// TIA Portal project "Kağıt Ambalaj Konik PLC (1,2,3,4,5)_V15.1" (V15.1)

(* hardware
DEVICE "S7-1200 station_1"  S7-1200 Station
   slot 0: "Rack_0"  S7-1200 Rack  Rack  V1.0
   slot 1: "PLC_1"  CPU 1215C DC/DC/DC  6ES7 215-1AG40-0XB0  V4.2
   slot 2: "DI 16x24VDC_1"  6ES7 221-1BH32-0XB0  V2.0
   slot 3: "AI 8x13BIT_1"  6ES7 231-4HF32-0XB0  V2.0
*)

// ===== PLC "PLC_1"  CPU 1215C DC/DC/DC =====

VAR_GLOBAL   // PLC tag table "Default tag table"
   "Konik 5 Count Value" AT %ID1000 : DWord;
   "Konik 4 Count Value" AT %ID1004 : DWord;
   "Konik 3 Count Value" AT %ID1008 : DWord;
   "Konik 2 Count Value" AT %ID1012 : DWord;
   "Konik 1 Count Value" AT %ID1016 : DWord;
   "Konik 1 Adet Sayaç" AT %I8.4 : Bool;
   "Konik 2 Adet Sayaç" AT %I8.5 : Bool;
   "System_Byte" AT %MB1 : Byte;
   "FirstScan" AT %M1.0 : Bool;
   "DiagStatusUpdate" AT %M1.1 : Bool;
   "AlwaysTRUE" AT %M1.2 : Bool;
   "AlwaysFALSE" AT %M1.3 : Bool;
   "Clock_Byte" AT %MB0 : Byte;
   "Clock_10Hz" AT %M0.0 : Bool;
   "Clock_5Hz" AT %M0.1 : Bool;
   "Clock_2.5Hz" AT %M0.2 : Bool;
   "Clock_2Hz" AT %M0.3 : Bool;
   "Clock_1.25Hz" AT %M0.4 : Bool;
   "Clock_1Hz" AT %M0.5 : Bool;
   "Clock_0.625Hz" AT %M0.6 : Bool;
   "Clock_0.5Hz" AT %M0.7 : Bool;
   "Konik 4 Adet Sayaç" AT %I9.1 : Bool;
   "Konik 5 Adet Sayaç" AT %I9.2 : Bool;
   "Konik 1 Run Bilgisi" AT %I9.3 : Bool;
   "Konik 2 Run Bilgisi" AT %I9.4 : Bool;
   "Konik 3 Run Bilgisi" AT %I9.5 : Bool;
   "Konik 4 Run Bilgisi" AT %I9.6 : Bool;
   "Konik 5 Run Bilgisi" AT %I9.7 : Bool;
   "Konik 3 Adet Sayaç" AT %I9.0 : Bool;
   "Tag_1" AT %M20.0 : Bool;
   "Tag_2" AT %M20.1 : Bool;
   "Tag_3" AT %M20.3 : Bool;
   "Tag_4" AT %M20.4 : Bool;
   "Tag_5" AT %M20.5 : Bool;
   "Tag_6" AT %M20.6 : Bool;
   "Tag_7" AT %M20.7 : Bool;
   "Tag_8" AT %M21.0 : Bool;
   "Tag_test" AT %I0.5 : Bool;
END_VAR

VAR_GLOBAL   // PLC tag table "Tag table_1"
   "Tag_rst_1" AT %M21.1 : Bool;
   "Tag_rst_2" AT %M21.2 : Bool;
   "Tag_rst_3" AT %M21.3 : Bool;
   "Tag_rst_4" AT %M21.5 : Bool;
   "Tag_rst_5" AT %M21.6 : Bool;
   "Tag_rst_6" AT %M21.7 : Bool;
   "Tag_rst_7" AT %M22.0 : Bool;
   "Tag_rst_8" AT %M22.1 : Bool;
   "Tag_rst_9" AT %M22.4 : Bool;
   "Tag_rst_10" AT %M22.5 : Bool;
   "Tag_rst_11" AT %M22.6 : Bool;
   "Tag_rst_12" AT %M22.7 : Bool;
   "Tag_rst_13" AT %M22.3 : Bool;
   "Tag_rst_14" AT %M22.2 : Bool;
   "Tag_rst_15" AT %M21.4 : Bool;
   "Tag_rst_16" AT %M23.0 : Bool;
   "Tag_rst_17" AT %M23.1 : Bool;
   "Tag_rst_18" AT %M23.2 : Bool;
   "Tag_rst_19" AT %M23.3 : Bool;
   "Tag_rst_20" AT %M23.4 : Bool;
   "Tag_rst_21" AT %M23.5 : Bool;
   "Tag_rst_22" AT %M23.6 : Bool;
   "Tag_rst_23" AT %M23.7 : Bool;
   "Tag_rst_24" AT %M24.0 : Bool;
   "hızcontrol" AT %M24.1 : Bool;
   "hızcontrol(1)" AT %M24.2 : Bool;
   "hızcontrol(2)" AT %M24.3 : Bool;
   "hızcontrol(3)" AT %M24.4 : Bool;
   "hızcontrol(4)" AT %M24.5 : Bool;
END_VAR

DATA_BLOCK "DataMeter"   // DB3
{ S7_Optimized_Access := 'FALSE' }
VERSION : 0.1
   VAR
      "Konik 1 Metre Sayac" : UDInt;
      "Konik 2 Metre Sayac" : UDInt;
      "Konik 3 Metre Sayac" : UDInt;
      "Konik 4 Metre Sayac" : UDInt;
      "Konik 5 Metre Sayac" : UDInt;
      "Konik 1 Metre RST" : Bool;
      "Konik 2 Metre RST" : Bool;
      "Konik 3 Metre RST" : Bool;
      "Konik 4 Metre RST" : Bool;
      "Konik 5 Metre RST" : Bool;
      "Konik 1 Hız" : Real;
      "Konik 2 Hız" : Real;
      "Konik 3 Hız" : Real;
      "Konik 4 Hız" : Real;
      "Konik 5 Hız" : Real;
      MultiplierValue : Real := 0.39284;
      EncoderRawValues : Array[0..4] of UDInt;
      TempMeters : Array[0..9] of UDInt;
      Rawspeed : Array[0..7] of Real;
      RealMeterValue : Array[0..7] of Real;
   END_VAR
BEGIN
END_DATA_BLOCK

DATA_BLOCK "DataSteam"   // DB4
{ S7_Optimized_Access := 'FALSE' }
VERSION : 0.1
   VAR
      sayıcıtest : UDInt := 0;
      wordtest : Word;
      udinttest : UDInt;
      dinttest : DInt;
      inttest_1 : Int;
      floattest : Real;
   END_VAR
BEGIN
END_DATA_BLOCK

DATA_BLOCK "DataDI"   // DB5
{ S7_Optimized_Access := 'FALSE' }
VERSION : 0.1
   VAR
      "Konik 1 Üretim sayacı" : UDInt;
      "Konik 2 Üretim sayacı" : UDInt;
      "Konik 3 Üretim sayacı" : UDInt;
      "Konik 4 Üretim sayacı" : UDInt;
      "Konik 5 Üretim sayacı" : UDInt;
      "Konik 1 Besleme Run Sinyal" : Bool;
      "Konik 2 Besleme Run Sinyal" : Bool;
      "Konik 3  BeslemeRun Sinyal" : Bool;
      "Konik 4  BeslemeRun Sinyal" : Bool;
      "Konik 5  BeslemeRun Sinyal" : Bool;
      "Konik 1 Sayac RST" : Bool;
      "Konik 2 Sayac RST" : Bool;
      "Konik 3 Sayac RST" : Bool;
      "Konik 4 Sayac RST" : Bool;
      "Konik 5 Sayac RST" : Bool;
      "Konik 1 Üretim Sayac Hızı" : Int;
      "Konik 2 Üretim Sayac Hızı" : Int;
      "Konik 3 Üretim Sayac Hızı" : Int;
      "Konik 4 Üretim Sayac Hızı" : Int;
      "Konik 5 Üretim Sayac Hızı" : Int;
      "Konik 1 Run Sinyal" : Bool;
      "Konik 2 Run Sinyal" : Bool;
      "Konik 3 Run Sinyal" : Bool;
      "Konik 4 Run Sinyal" : Bool;
      "Konik 5 Run Sinyal" : Bool;
      "Konik RST" : Array[0..9] of Bool;
      "Konik adet temp" : Array[0..9] of UDInt;
      Dakikareset : Bool;
   END_VAR
BEGIN
END_DATA_BLOCK

DATA_BLOCK "DataSendDI"   // DB6
{ S7_Optimized_Access := 'FALSE' }
VERSION : 0.1
   VAR
      "Konik 1 Run Sinyal" : Bool;
      "Konik 2 Run Sinyal" : Bool;
      "Konik 3 Run Sinyal" : Bool;
      "Konik 4 Run Sinyal" : Bool;
      "Konik 5 Run Sinyal" : Bool;
      "Konik 1 Sayac RST" : Bool;
      "Konik 2 Sayac RST" : Bool;
      "Konik 3 Sayac RST" : Bool;
      "Konik 4 Sayac RST" : Bool;
      "Konik 5 Sayac RST" : Bool;
      "Konik 1 Besleme Run Sinyal" : Bool;
      "Konik 2 Besleme Run Sinyal" : Bool;
      "Konik 3  BeslemeRun Sinyal" : Bool;
      "Konik 4  BeslemeRun Sinyal" : Bool;
      "Konik 5  BeslemeRun Sinyal" : Bool;
      "Konik 1 Metre RST" : Bool;
      "Konik 3 Metre RST" : Bool;
      "Konik 4 Metre RST" : Bool;
      "Konik 5 Metre RST" : Bool;
      "Konik 2 Metre RST" : Bool;
      "Konik 1 Üretim sayacı" : Real;
      "Konik 2 Üretim sayacı" : Real;
      "Konik 3 Üretim sayacı" : Real;
      "Konik 4 Üretim sayacı" : Real;
      "Konik 5 Üretim sayacı" : Real;
      "Konik 1 Üretim Sayac Hızı" : Real;
      "Konik 2 Üretim Sayac Hızı" : Real;
      "Konik 3 Üretim Sayac Hızı" : Real;
      "Konik 4 Üretim Sayac Hızı" : Real;
      "Konik 5 Üretim Sayac Hızı" : Real;
      "Konik 1 Metre Sayac" : Real;
      "Konik 2 Metre Sayac" : Real;
      "Konik 3 Metre Sayac" : Real;
      "Konik 4 Metre Sayac" : Real;
      "Konik 5 Metre Sayac" : Real;
      "Konik 1 Hız" : Real;
      "Konik 2 Hız" : Real;
      "Konik 3 Hız" : Real;
      "Konik 4 Hız" : Real;
      "Konik 5 Hız" : Real;
      PLCLiveBit : Real;
   END_VAR
BEGIN
END_DATA_BLOCK

// folder: System blocks/Program resources

DATA_BLOCK "Counter_dakika"   // DB1
{ S7_Optimized_Access := 'TRUE' }
AUTHOR : Simatic
FAMILY : IEC
NAME : CNTR
VERSION : 1.0
// stored: InstanceOfName IEC_COUNTER
"IEC_COUNTER"
BEGIN
END_DATA_BLOCK

DATA_BLOCK "IEC_Counter_0_DB_5"   // DB2
{ S7_Optimized_Access := 'TRUE' }
AUTHOR : Simatic
FAMILY : IEC
NAME : UDCNTR
VERSION : 1.2
// stored: InstanceOfName IEC_UDCOUNTER
"IEC_UDCOUNTER"
BEGIN
END_DATA_BLOCK

DATA_BLOCK "livetimer"   // DB7
{ S7_Optimized_Access := 'TRUE' }
AUTHOR : Simatic
FAMILY : IEC
NAME : IEC_TMR
VERSION : 1.0
// stored: InstanceOfName IEC_TIMER
"IEC_TIMER"
BEGIN
END_DATA_BLOCK

DATA_BLOCK "IEC_Counter_0_DB"   // DB30
{ S7_Optimized_Access := 'TRUE' }
AUTHOR : Simatic
FAMILY : IEC
NAME : UDCNTR
VERSION : 1.2
// stored: InstanceOfName IEC_UDCOUNTER
"IEC_UDCOUNTER"
BEGIN
END_DATA_BLOCK

DATA_BLOCK "IEC_Counter_0_DB_1"   // DB31
{ S7_Optimized_Access := 'TRUE' }
AUTHOR : Simatic
FAMILY : IEC
NAME : UDCNTR
VERSION : 1.2
// stored: InstanceOfName IEC_UDCOUNTER
"IEC_UDCOUNTER"
BEGIN
END_DATA_BLOCK

DATA_BLOCK "IEC_Counter_0_DB_2"   // DB32
{ S7_Optimized_Access := 'TRUE' }
AUTHOR : Simatic
FAMILY : IEC
NAME : UDCNTR
VERSION : 1.2
// stored: InstanceOfName IEC_UDCOUNTER
"IEC_UDCOUNTER"
BEGIN
END_DATA_BLOCK

DATA_BLOCK "IEC_Counter_0_DB_3"   // DB33
{ S7_Optimized_Access := 'TRUE' }
AUTHOR : Simatic
FAMILY : IEC
NAME : UDCNTR
VERSION : 1.2
// stored: InstanceOfName IEC_UDCOUNTER
"IEC_UDCOUNTER"
BEGIN
END_DATA_BLOCK

DATA_BLOCK "IEC_Counter_0_DB_4"   // DB34
{ S7_Optimized_Access := 'TRUE' }
AUTHOR : Simatic
FAMILY : IEC
NAME : UDCNTR
VERSION : 1.2
// stored: InstanceOfName IEC_UDCOUNTER
"IEC_UDCOUNTER"
BEGIN
END_DATA_BLOCK

// folder: (top level)

FUNCTION "EncoderSingleton" : Void   // FC1, LAD
{ S7_Optimized_Access := 'TRUE' }
VERSION : 0.1
   VAR_TEMP   // added for the SCL form of the ladder/FBD networks
      _w1 : Bool;
      _w2 : Bool;
      _w3 : Bool;
      _w4 : Bool;
      _w5 : Bool;
   END_VAR
BEGIN

REGION Network 1: HSC INIT
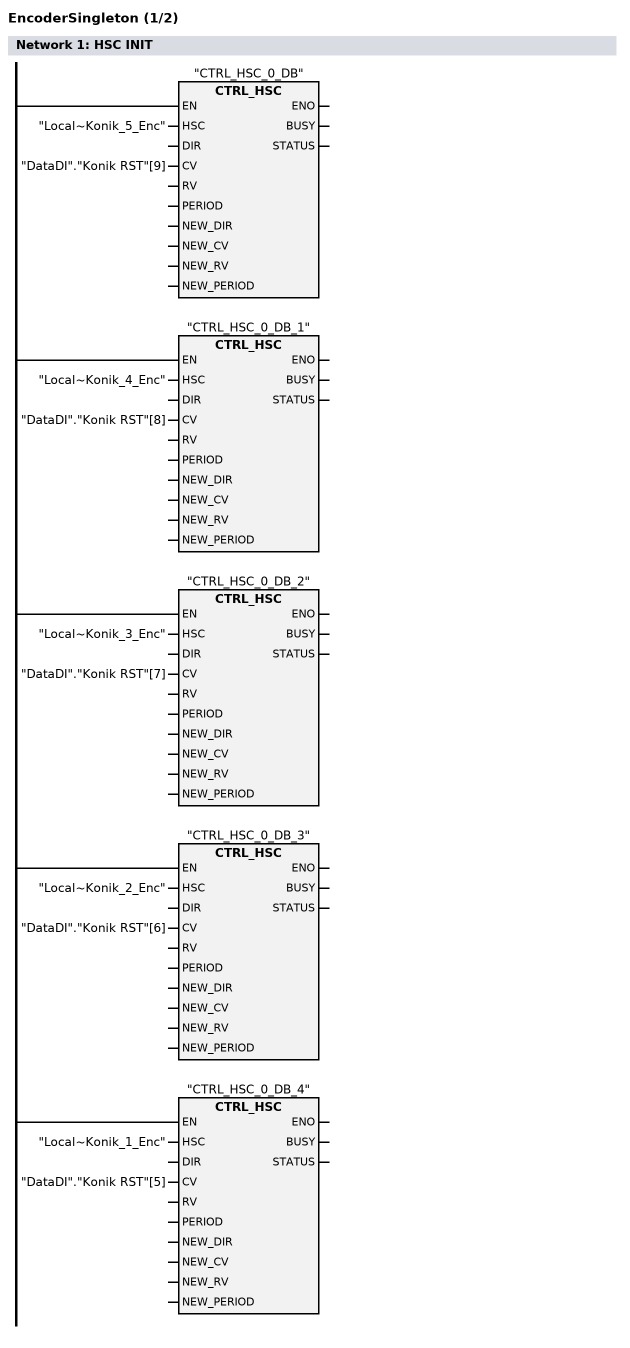
   "CTRL_HSC_0_DB"(HSC := "Local~Konik_5_Enc", CV := "DataDI"."Konik RST"[9]);   // CTRL_HSC
   "CTRL_HSC_0_DB_1"(HSC := "Local~Konik_4_Enc", CV := "DataDI"."Konik RST"[8]);   // CTRL_HSC
   "CTRL_HSC_0_DB_2"(HSC := "Local~Konik_3_Enc", CV := "DataDI"."Konik RST"[7]);   // CTRL_HSC
   "CTRL_HSC_0_DB_3"(HSC := "Local~Konik_2_Enc", CV := "DataDI"."Konik RST"[6]);   // CTRL_HSC
   "CTRL_HSC_0_DB_4"(HSC := "Local~Konik_1_Enc", CV := "DataDI"."Konik RST"[5]);   // CTRL_HSC
END_REGION

REGION Network 2
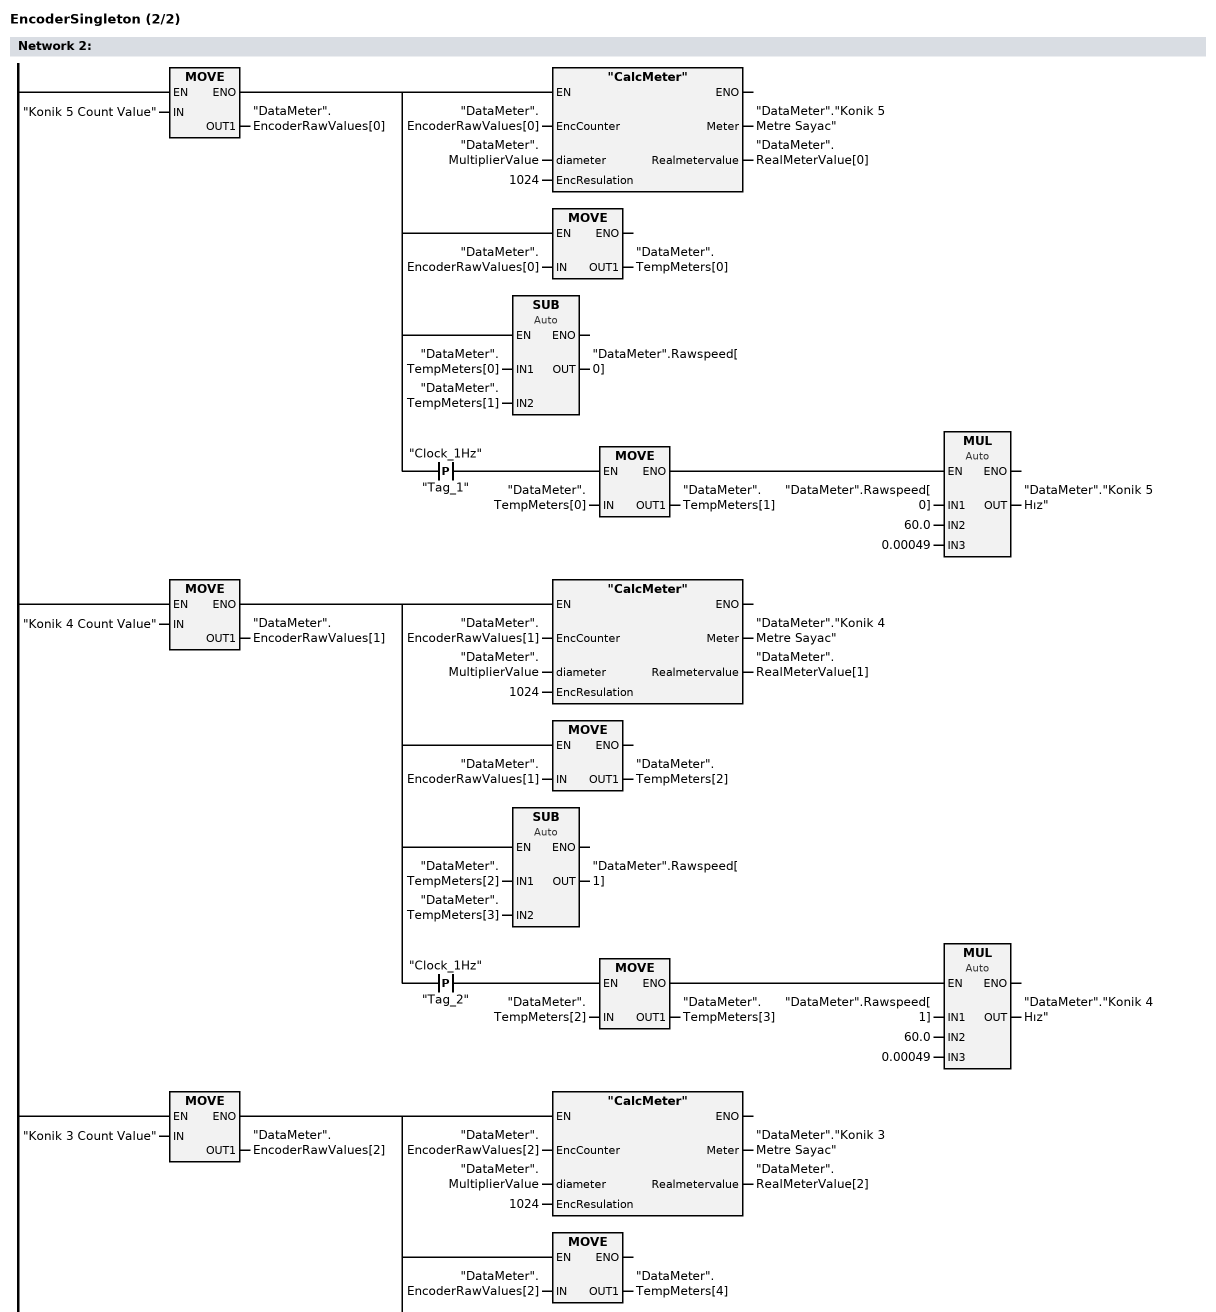
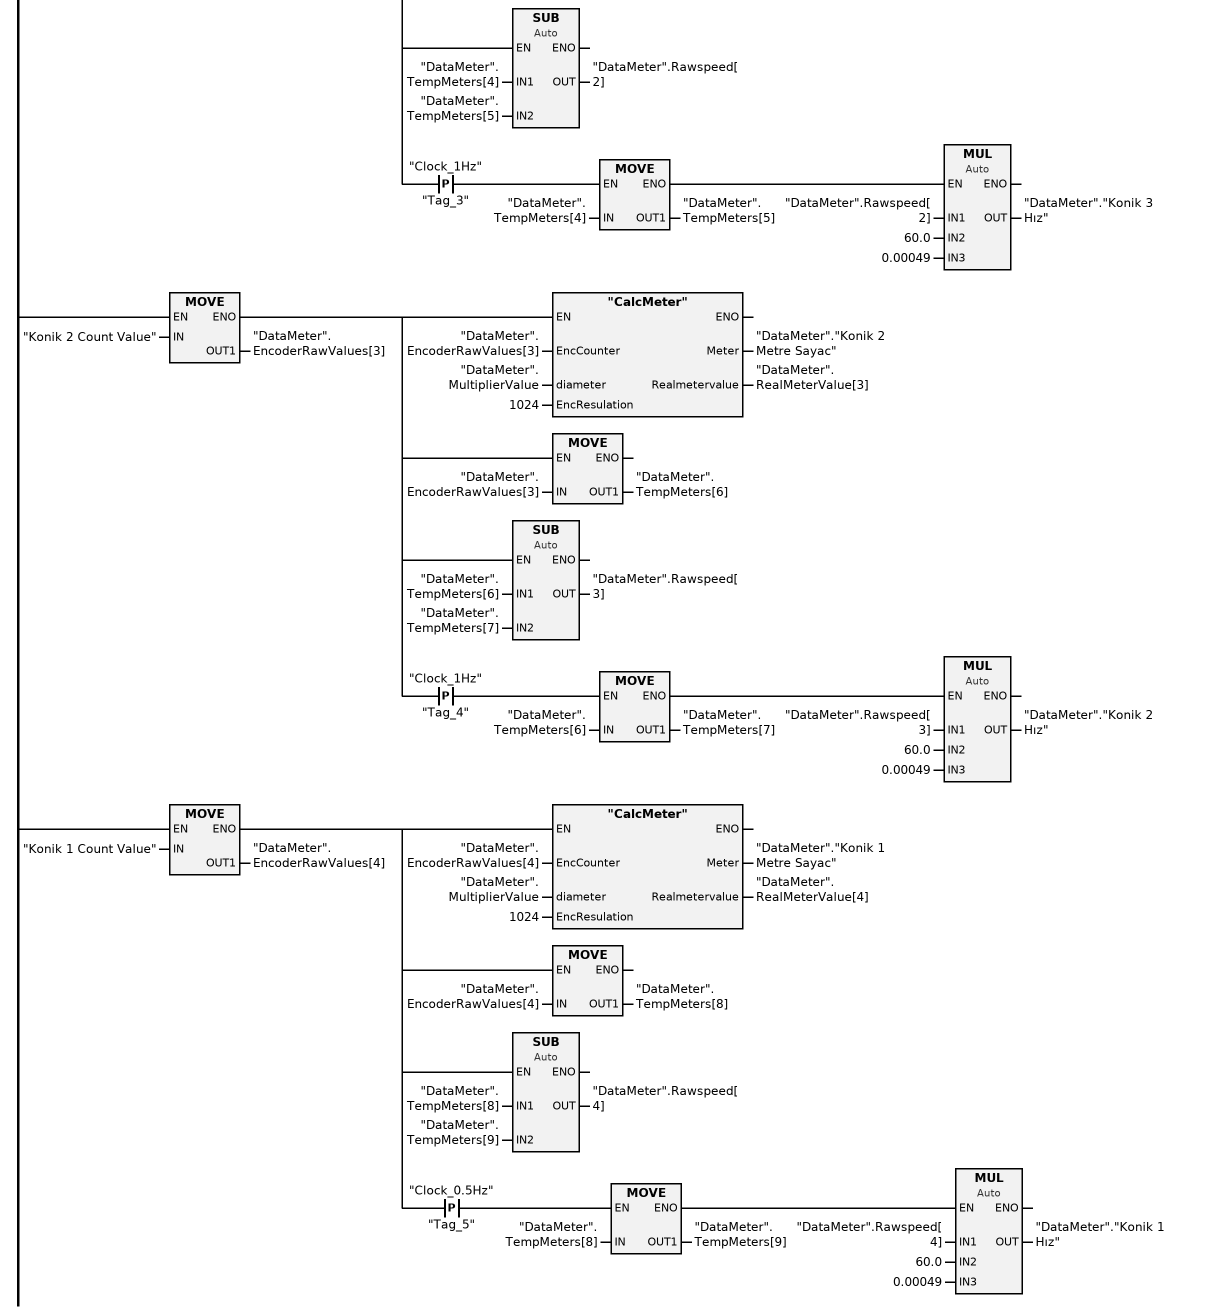
   RUNG wire#powerrail
      Move(in := "Konik 5 Count Value", out1 => "DataMeter".EncoderRawValues[0])
      wire#w1
      "CalcMeter"(EncCounter := "DataMeter".EncoderRawValues[0], diameter := "DataMeter".MultiplierValue, EncResulation := 1024, Meter => "DataMeter"."Konik 5 Metre Sayac", Realmetervalue => "DataMeter".RealMeterValue[0])
   END_RUNG
   RUNG wire#w1
      Move(in := "DataMeter".EncoderRawValues[0], out1 => "DataMeter".TempMeters[0])
   END_RUNG
   RUNG wire#w1
      Sub(in1 := "DataMeter".TempMeters[0], in2 := "DataMeter".TempMeters[1], out => "DataMeter".Rawspeed[0])
   END_RUNG
   RUNG wire#w1
      P_Contact(operand := "Clock_1Hz", bit := "Tag_1")
      Move(in := "DataMeter".TempMeters[0], out1 => "DataMeter".TempMeters[1])
      Mul(in1 := "DataMeter".Rawspeed[0], in2 := 60.0, in3 := 0.00049, out => "DataMeter"."Konik 5 Hız")
   END_RUNG
   RUNG wire#powerrail
      Move(in := "Konik 4 Count Value", out1 => "DataMeter".EncoderRawValues[1])
      wire#w2
      "CalcMeter"(EncCounter := "DataMeter".EncoderRawValues[1], diameter := "DataMeter".MultiplierValue, EncResulation := 1024, Meter => "DataMeter"."Konik 4 Metre Sayac", Realmetervalue => "DataMeter".RealMeterValue[1])
   END_RUNG
   RUNG wire#w2
      Move(in := "DataMeter".EncoderRawValues[1], out1 => "DataMeter".TempMeters[2])
   END_RUNG
   RUNG wire#w2
      Sub(in1 := "DataMeter".TempMeters[2], in2 := "DataMeter".TempMeters[3], out => "DataMeter".Rawspeed[1])
   END_RUNG
   RUNG wire#w2
      P_Contact(operand := "Clock_1Hz", bit := "Tag_2")
      Move(in := "DataMeter".TempMeters[2], out1 => "DataMeter".TempMeters[3])
      Mul(in1 := "DataMeter".Rawspeed[1], in2 := 60.0, in3 := 0.00049, out => "DataMeter"."Konik 4 Hız")
   END_RUNG
   RUNG wire#powerrail
      Move(in := "Konik 3 Count Value", out1 => "DataMeter".EncoderRawValues[2])
      wire#w3
      "CalcMeter"(EncCounter := "DataMeter".EncoderRawValues[2], diameter := "DataMeter".MultiplierValue, EncResulation := 1024, Meter => "DataMeter"."Konik 3 Metre Sayac", Realmetervalue => "DataMeter".RealMeterValue[2])
   END_RUNG
   RUNG wire#w3
      Move(in := "DataMeter".EncoderRawValues[2], out1 => "DataMeter".TempMeters[4])
   END_RUNG
   RUNG wire#w3
      Sub(in1 := "DataMeter".TempMeters[4], in2 := "DataMeter".TempMeters[5], out => "DataMeter".Rawspeed[2])
   END_RUNG
   RUNG wire#w3
      P_Contact(operand := "Clock_1Hz", bit := "Tag_3")
      Move(in := "DataMeter".TempMeters[4], out1 => "DataMeter".TempMeters[5])
      Mul(in1 := "DataMeter".Rawspeed[2], in2 := 60.0, in3 := 0.00049, out => "DataMeter"."Konik 3 Hız")
   END_RUNG
   RUNG wire#powerrail
      Move(in := "Konik 2 Count Value", out1 => "DataMeter".EncoderRawValues[3])
      wire#w4
      "CalcMeter"(EncCounter := "DataMeter".EncoderRawValues[3], diameter := "DataMeter".MultiplierValue, EncResulation := 1024, Meter => "DataMeter"."Konik 2 Metre Sayac", Realmetervalue => "DataMeter".RealMeterValue[3])
   END_RUNG
   RUNG wire#w4
      Move(in := "DataMeter".EncoderRawValues[3], out1 => "DataMeter".TempMeters[6])
   END_RUNG
   RUNG wire#w4
      Sub(in1 := "DataMeter".TempMeters[6], in2 := "DataMeter".TempMeters[7], out => "DataMeter".Rawspeed[3])
   END_RUNG
   RUNG wire#w4
      P_Contact(operand := "Clock_1Hz", bit := "Tag_4")
      Move(in := "DataMeter".TempMeters[6], out1 => "DataMeter".TempMeters[7])
      Mul(in1 := "DataMeter".Rawspeed[3], in2 := 60.0, in3 := 0.00049, out => "DataMeter"."Konik 2 Hız")
   END_RUNG
   RUNG wire#powerrail
      Move(in := "Konik 1 Count Value", out1 => "DataMeter".EncoderRawValues[4])
      wire#w5
      "CalcMeter"(EncCounter := "DataMeter".EncoderRawValues[4], diameter := "DataMeter".MultiplierValue, EncResulation := 1024, Meter => "DataMeter"."Konik 1 Metre Sayac", Realmetervalue => "DataMeter".RealMeterValue[4])
   END_RUNG
   RUNG wire#w5
      Move(in := "DataMeter".EncoderRawValues[4], out1 => "DataMeter".TempMeters[8])
   END_RUNG
   RUNG wire#w5
      Sub(in1 := "DataMeter".TempMeters[8], in2 := "DataMeter".TempMeters[9], out => "DataMeter".Rawspeed[4])
   END_RUNG
   RUNG wire#w5
      P_Contact(operand := "Clock_0.5Hz", bit := "Tag_5")
      Move(in := "DataMeter".TempMeters[8], out1 => "DataMeter".TempMeters[9])
      Mul(in1 := "DataMeter".Rawspeed[4], in2 := 60.0, in3 := 0.00049, out => "DataMeter"."Konik 1 Hız")
   END_RUNG
   // the same network as SCL:
   "DataMeter".EncoderRawValues[0] := "Konik 5 Count Value";
   "CalcMeter"(EncCounter := "DataMeter".EncoderRawValues[0],
               diameter := "DataMeter".MultiplierValue,
               EncResulation := 1024,
               Meter => "DataMeter"."Konik 5 Metre Sayac",
               Realmetervalue => "DataMeter".RealMeterValue[0]);
   "DataMeter".TempMeters[0] := "DataMeter".EncoderRawValues[0];
   "DataMeter".Rawspeed[0] := "DataMeter".TempMeters[0] - "DataMeter".TempMeters[1];
   #_w1 := "Clock_1Hz" AND NOT "Tag_1";   // rising edge of "Clock_1Hz"
   "Tag_1" := "Clock_1Hz";
   IF #_w1 THEN
       "DataMeter".TempMeters[1] := "DataMeter".TempMeters[0];
       "DataMeter"."Konik 5 Hız" := "DataMeter".Rawspeed[0] * 60.0 * 0.00049;
   END_IF;
   "DataMeter".EncoderRawValues[1] := "Konik 4 Count Value";
   "CalcMeter"(EncCounter := "DataMeter".EncoderRawValues[1],
               diameter := "DataMeter".MultiplierValue,
               EncResulation := 1024,
               Meter => "DataMeter"."Konik 4 Metre Sayac",
               Realmetervalue => "DataMeter".RealMeterValue[1]);
   "DataMeter".TempMeters[2] := "DataMeter".EncoderRawValues[1];
   "DataMeter".Rawspeed[1] := "DataMeter".TempMeters[2] - "DataMeter".TempMeters[3];
   #_w2 := "Clock_1Hz" AND NOT "Tag_2";   // rising edge of "Clock_1Hz"
   "Tag_2" := "Clock_1Hz";
   IF #_w2 THEN
       "DataMeter".TempMeters[3] := "DataMeter".TempMeters[2];
       "DataMeter"."Konik 4 Hız" := "DataMeter".Rawspeed[1] * 60.0 * 0.00049;
   END_IF;
   "DataMeter".EncoderRawValues[2] := "Konik 3 Count Value";
   "CalcMeter"(EncCounter := "DataMeter".EncoderRawValues[2],
               diameter := "DataMeter".MultiplierValue,
               EncResulation := 1024,
               Meter => "DataMeter"."Konik 3 Metre Sayac",
               Realmetervalue => "DataMeter".RealMeterValue[2]);
   "DataMeter".TempMeters[4] := "DataMeter".EncoderRawValues[2];
   "DataMeter".Rawspeed[2] := "DataMeter".TempMeters[4] - "DataMeter".TempMeters[5];
   #_w3 := "Clock_1Hz" AND NOT "Tag_3";   // rising edge of "Clock_1Hz"
   "Tag_3" := "Clock_1Hz";
   IF #_w3 THEN
       "DataMeter".TempMeters[5] := "DataMeter".TempMeters[4];
       "DataMeter"."Konik 3 Hız" := "DataMeter".Rawspeed[2] * 60.0 * 0.00049;
   END_IF;
   "DataMeter".EncoderRawValues[3] := "Konik 2 Count Value";
   "CalcMeter"(EncCounter := "DataMeter".EncoderRawValues[3],
               diameter := "DataMeter".MultiplierValue,
               EncResulation := 1024,
               Meter => "DataMeter"."Konik 2 Metre Sayac",
               Realmetervalue => "DataMeter".RealMeterValue[3]);
   "DataMeter".TempMeters[6] := "DataMeter".EncoderRawValues[3];
   "DataMeter".Rawspeed[3] := "DataMeter".TempMeters[6] - "DataMeter".TempMeters[7];
   #_w4 := "Clock_1Hz" AND NOT "Tag_4";   // rising edge of "Clock_1Hz"
   "Tag_4" := "Clock_1Hz";
   IF #_w4 THEN
       "DataMeter".TempMeters[7] := "DataMeter".TempMeters[6];
       "DataMeter"."Konik 2 Hız" := "DataMeter".Rawspeed[3] * 60.0 * 0.00049;
   END_IF;
   "DataMeter".EncoderRawValues[4] := "Konik 1 Count Value";
   "CalcMeter"(EncCounter := "DataMeter".EncoderRawValues[4],
               diameter := "DataMeter".MultiplierValue,
               EncResulation := 1024,
               Meter => "DataMeter"."Konik 1 Metre Sayac",
               Realmetervalue => "DataMeter".RealMeterValue[4]);
   "DataMeter".TempMeters[8] := "DataMeter".EncoderRawValues[4];
   "DataMeter".Rawspeed[4] := "DataMeter".TempMeters[8] - "DataMeter".TempMeters[9];
   #_w5 := "Clock_0.5Hz" AND NOT "Tag_5";   // rising edge of "Clock_0.5Hz"
   "Tag_5" := "Clock_0.5Hz";
   IF #_w5 THEN
       "DataMeter".TempMeters[9] := "DataMeter".TempMeters[8];
       "DataMeter"."Konik 1 Hız" := "DataMeter".Rawspeed[4] * 60.0 * 0.00049;
   END_IF;
END_REGION
END_FUNCTION

FUNCTION "SteamSingleton" : Void   // FC2, LAD
{ S7_Optimized_Access := 'TRUE' }
VERSION : 0.1
BEGIN
END_FUNCTION

FUNCTION "DISingleton" : Void   // FC3, LAD
{ S7_Optimized_Access := 'TRUE' }
VERSION : 0.1
BEGIN

REGION Network 1: Cisim Adet Sayaçları
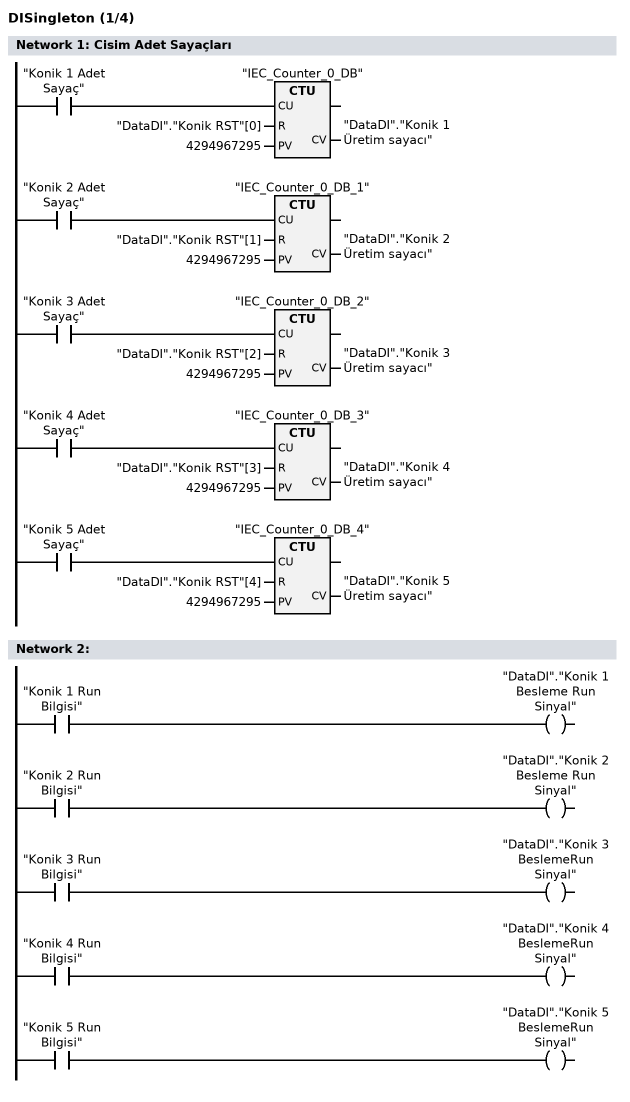
   "IEC_Counter_0_DB".CTU(CU := "Konik 1 Adet Sayaç",
                          R := "DataDI"."Konik RST"[0],
                          PV := 4294967295,
                          CV => "DataDI"."Konik 1 Üretim sayacı");
   "IEC_Counter_0_DB_1".CTU(CU := "Konik 2 Adet Sayaç",
                           R := "DataDI"."Konik RST"[1],
                           PV := 4294967295,
                           CV => "DataDI"."Konik 2 Üretim sayacı");
   "IEC_Counter_0_DB_2".CTU(CU := "Konik 3 Adet Sayaç",
                           R := "DataDI"."Konik RST"[2],
                           PV := 4294967295,
                           CV => "DataDI"."Konik 3 Üretim sayacı");
   "IEC_Counter_0_DB_3".CTU(CU := "Konik 4 Adet Sayaç",
                           R := "DataDI"."Konik RST"[3],
                           PV := 4294967295,
                           CV => "DataDI"."Konik 4 Üretim sayacı");
   "IEC_Counter_0_DB_4".CTU(CU := "Konik 5 Adet Sayaç",
                           R := "DataDI"."Konik RST"[4],
                           PV := 4294967295,
                           CV => "DataDI"."Konik 5 Üretim sayacı");
END_REGION

REGION Network 2
   RUNG wire#powerrail
      Contact( "Konik 1 Run Bilgisi" )
      Coil( "DataDI"."Konik 1 Besleme Run Sinyal" )
   END_RUNG
   RUNG wire#powerrail
      Contact( "Konik 2 Run Bilgisi" )
      Coil( "DataDI"."Konik 2 Besleme Run Sinyal" )
   END_RUNG
   RUNG wire#powerrail
      Contact( "Konik 3 Run Bilgisi" )
      Coil( "DataDI"."Konik 3  BeslemeRun Sinyal" )
   END_RUNG
   RUNG wire#powerrail
      Contact( "Konik 4 Run Bilgisi" )
      Coil( "DataDI"."Konik 4  BeslemeRun Sinyal" )
   END_RUNG
   RUNG wire#powerrail
      Contact( "Konik 5 Run Bilgisi" )
      Coil( "DataDI"."Konik 5  BeslemeRun Sinyal" )
   END_RUNG
   // the same network as SCL:
   "DataDI"."Konik 1 Besleme Run Sinyal" := "Konik 1 Run Bilgisi";
   "DataDI"."Konik 2 Besleme Run Sinyal" := "Konik 2 Run Bilgisi";
   "DataDI"."Konik 3  BeslemeRun Sinyal" := "Konik 3 Run Bilgisi";
   "DataDI"."Konik 4  BeslemeRun Sinyal" := "Konik 4 Run Bilgisi";
   "DataDI"."Konik 5  BeslemeRun Sinyal" := "Konik 5 Run Bilgisi";
END_REGION

REGION Network 3
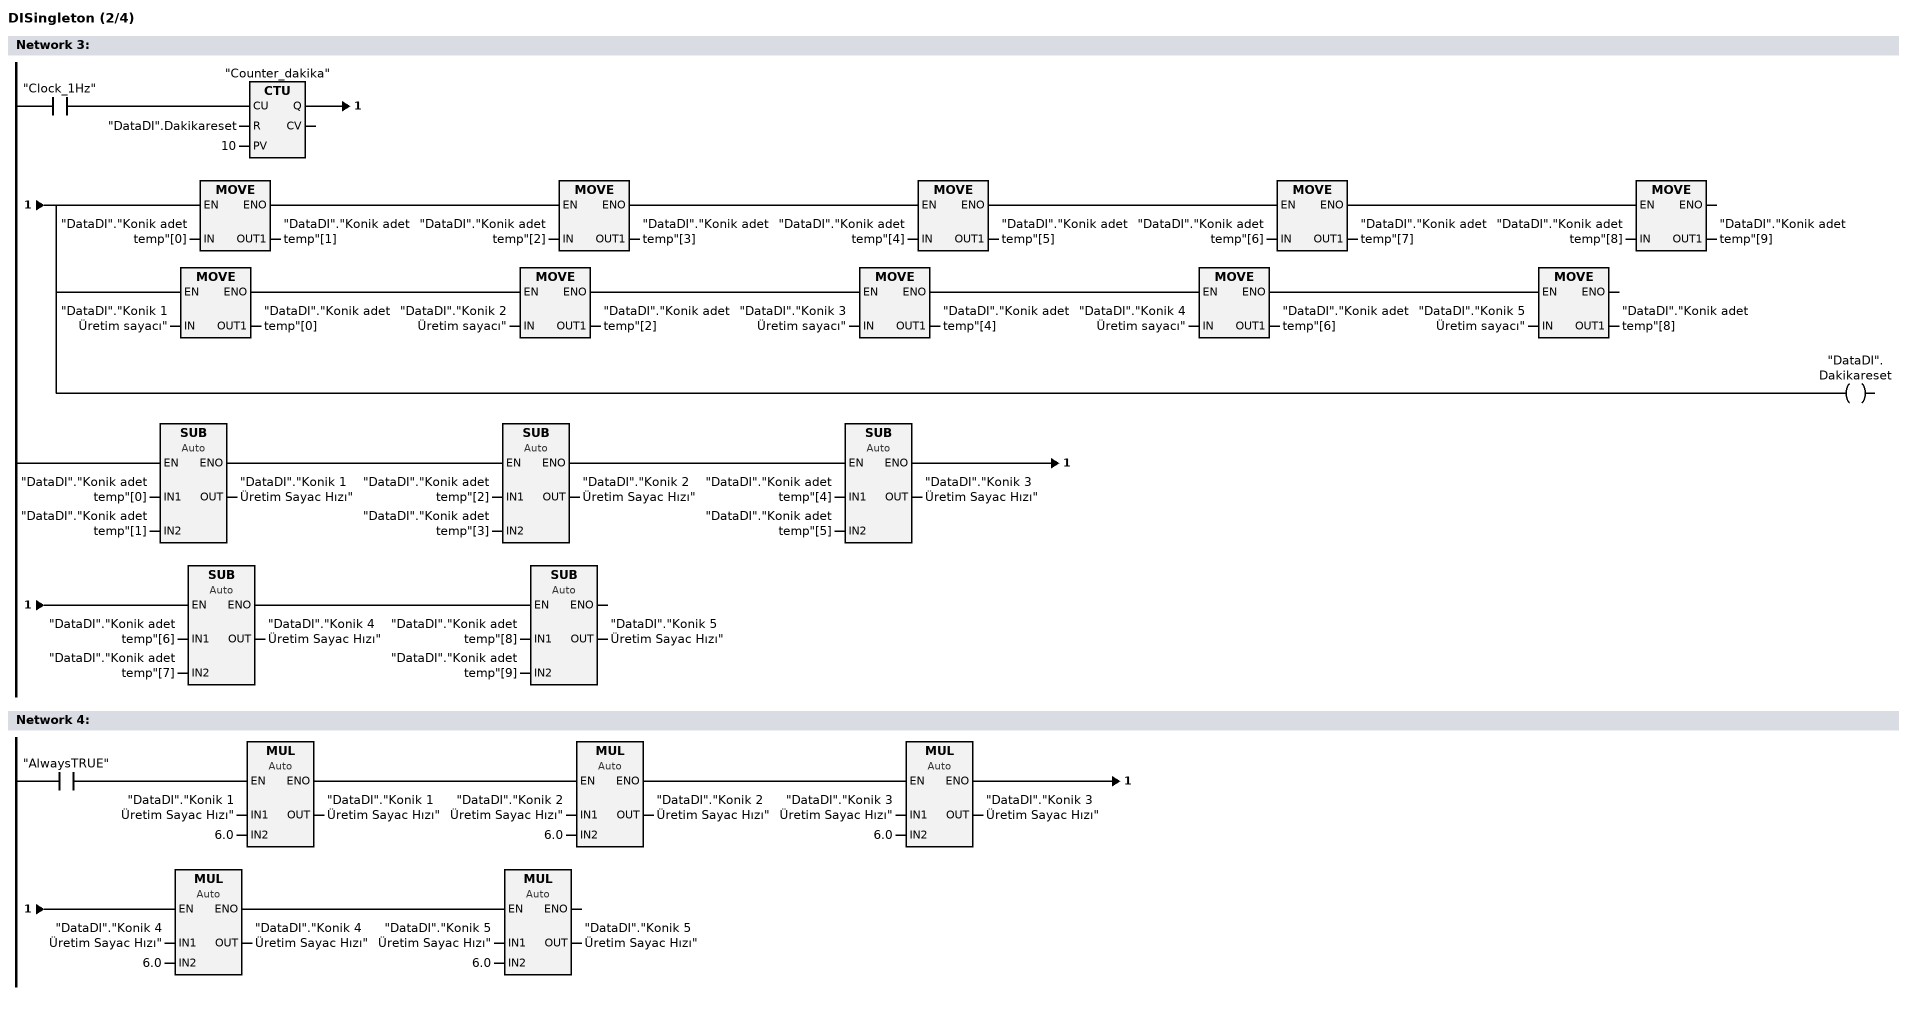
   "Counter_dakika".CTU(CU := "Clock_1Hz", R := "DataDI".Dakikareset, PV := 10);
   IF "Counter_dakika".Q THEN
       "DataDI"."Konik adet temp"[1] := "DataDI"."Konik adet temp"[0];
       "DataDI"."Konik adet temp"[3] := "DataDI"."Konik adet temp"[2];
       "DataDI"."Konik adet temp"[5] := "DataDI"."Konik adet temp"[4];
       "DataDI"."Konik adet temp"[7] := "DataDI"."Konik adet temp"[6];
       "DataDI"."Konik adet temp"[9] := "DataDI"."Konik adet temp"[8];
       "DataDI"."Konik adet temp"[0] := "DataDI"."Konik 1 Üretim sayacı";
       "DataDI"."Konik adet temp"[2] := "DataDI"."Konik 2 Üretim sayacı";
       "DataDI"."Konik adet temp"[4] := "DataDI"."Konik 3 Üretim sayacı";
       "DataDI"."Konik adet temp"[6] := "DataDI"."Konik 4 Üretim sayacı";
       "DataDI"."Konik adet temp"[8] := "DataDI"."Konik 5 Üretim sayacı";
   END_IF;
   "DataDI".Dakikareset := "Counter_dakika".Q;
   "DataDI"."Konik 1 Üretim Sayac Hızı" := "DataDI"."Konik adet temp"[0] - "DataDI"."Konik adet temp"[1];
   "DataDI"."Konik 2 Üretim Sayac Hızı" := "DataDI"."Konik adet temp"[2] - "DataDI"."Konik adet temp"[3];
   "DataDI"."Konik 3 Üretim Sayac Hızı" := "DataDI"."Konik adet temp"[4] - "DataDI"."Konik adet temp"[5];
   "DataDI"."Konik 4 Üretim Sayac Hızı" := "DataDI"."Konik adet temp"[6] - "DataDI"."Konik adet temp"[7];
   "DataDI"."Konik 5 Üretim Sayac Hızı" := "DataDI"."Konik adet temp"[8] - "DataDI"."Konik adet temp"[9];
END_REGION

REGION Network 4
   RUNG wire#powerrail
      Contact( "AlwaysTRUE" )
      Mul(in1 := "DataDI"."Konik 1 Üretim Sayac Hızı", in2 := 6.0, out => "DataDI"."Konik 1 Üretim Sayac Hızı")
      Mul(in1 := "DataDI"."Konik 2 Üretim Sayac Hızı", in2 := 6.0, out => "DataDI"."Konik 2 Üretim Sayac Hızı")
      Mul(in1 := "DataDI"."Konik 3 Üretim Sayac Hızı", in2 := 6.0, out => "DataDI"."Konik 3 Üretim Sayac Hızı")
      Mul(in1 := "DataDI"."Konik 4 Üretim Sayac Hızı", in2 := 6.0, out => "DataDI"."Konik 4 Üretim Sayac Hızı")
      Mul(in1 := "DataDI"."Konik 5 Üretim Sayac Hızı", in2 := 6.0, out => "DataDI"."Konik 5 Üretim Sayac Hızı")
   END_RUNG
   // the same network as SCL:
   IF "AlwaysTRUE" THEN
       "DataDI"."Konik 1 Üretim Sayac Hızı" := "DataDI"."Konik 1 Üretim Sayac Hızı" * 6.0;
       "DataDI"."Konik 2 Üretim Sayac Hızı" := "DataDI"."Konik 2 Üretim Sayac Hızı" * 6.0;
       "DataDI"."Konik 3 Üretim Sayac Hızı" := "DataDI"."Konik 3 Üretim Sayac Hızı" * 6.0;
       "DataDI"."Konik 4 Üretim Sayac Hızı" := "DataDI"."Konik 4 Üretim Sayac Hızı" * 6.0;
       "DataDI"."Konik 5 Üretim Sayac Hızı" := "DataDI"."Konik 5 Üretim Sayac Hızı" * 6.0;
   END_IF;
END_REGION

REGION Network 5
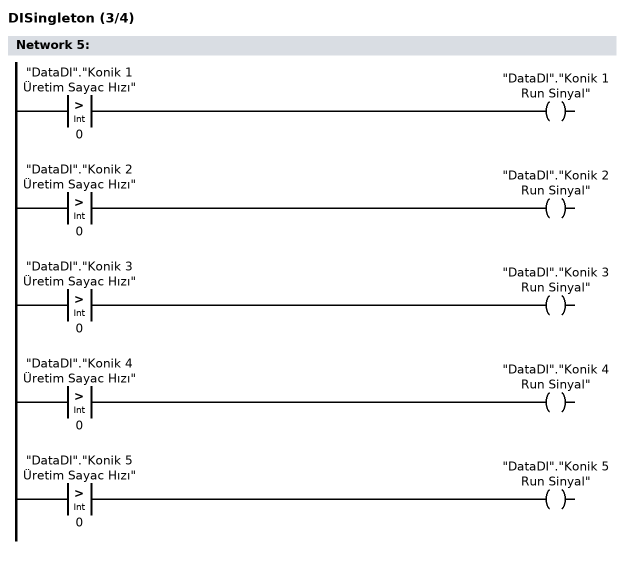
   RUNG wire#powerrail
      { S7_Templates := "SrcType := Int" } GT_Contact(in1 := "DataDI"."Konik 1 Üretim Sayac Hızı", in2 := 0)
      Coil( "DataDI"."Konik 1 Run Sinyal" )
   END_RUNG
   RUNG wire#powerrail
      { S7_Templates := "SrcType := Int" } GT_Contact(in1 := "DataDI"."Konik 2 Üretim Sayac Hızı", in2 := 0)
      Coil( "DataDI"."Konik 2 Run Sinyal" )
   END_RUNG
   RUNG wire#powerrail
      { S7_Templates := "SrcType := Int" } GT_Contact(in1 := "DataDI"."Konik 3 Üretim Sayac Hızı", in2 := 0)
      Coil( "DataDI"."Konik 3 Run Sinyal" )
   END_RUNG
   RUNG wire#powerrail
      { S7_Templates := "SrcType := Int" } GT_Contact(in1 := "DataDI"."Konik 4 Üretim Sayac Hızı", in2 := 0)
      Coil( "DataDI"."Konik 4 Run Sinyal" )
   END_RUNG
   RUNG wire#powerrail
      { S7_Templates := "SrcType := Int" } GT_Contact(in1 := "DataDI"."Konik 5 Üretim Sayac Hızı", in2 := 0)
      Coil( "DataDI"."Konik 5 Run Sinyal" )
   END_RUNG
   // the same network as SCL:
   "DataDI"."Konik 1 Run Sinyal" := "DataDI"."Konik 1 Üretim Sayac Hızı" > 0;
   "DataDI"."Konik 2 Run Sinyal" := "DataDI"."Konik 2 Üretim Sayac Hızı" > 0;
   "DataDI"."Konik 3 Run Sinyal" := "DataDI"."Konik 3 Üretim Sayac Hızı" > 0;
   "DataDI"."Konik 4 Run Sinyal" := "DataDI"."Konik 4 Üretim Sayac Hızı" > 0;
   "DataDI"."Konik 5 Run Sinyal" := "DataDI"."Konik 5 Üretim Sayac Hızı" > 0;
END_REGION

REGION Network 6
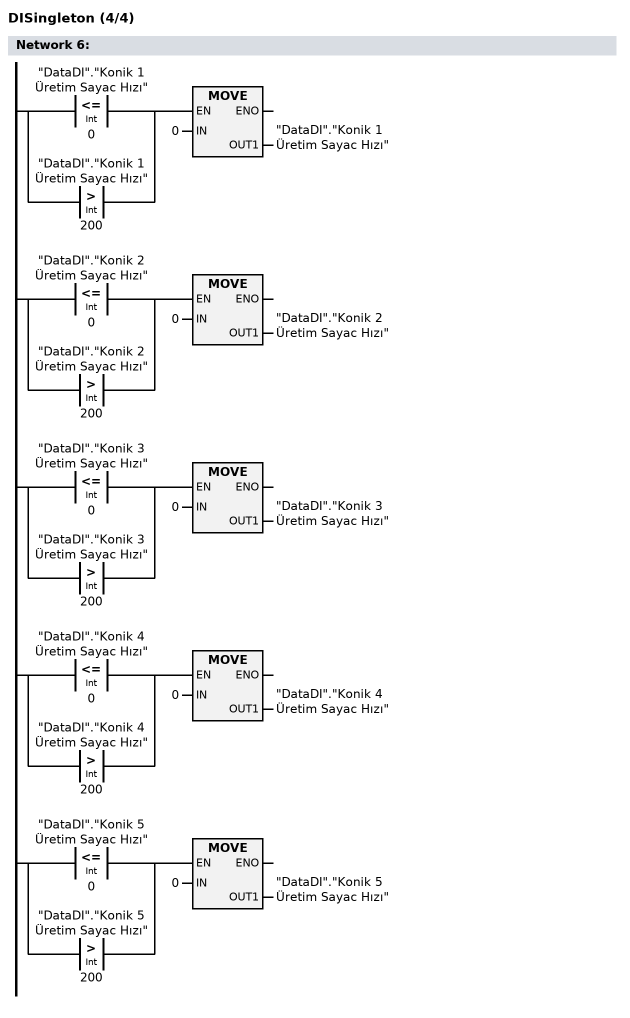
   RUNG wire#powerrail
      { S7_Templates := "SrcType := Int" } LE_Contact(in1 := "DataDI"."Konik 1 Üretim Sayac Hızı", in2 := 0)
      wire#w1
      Move(in := 0, out1 => "DataDI"."Konik 1 Üretim Sayac Hızı")
   END_RUNG
   RUNG wire#powerrail
      { S7_Templates := "SrcType := Int" } GT_Contact(in1 := "DataDI"."Konik 1 Üretim Sayac Hızı", in2 := 200)
   END_RUNG wire#w1
   RUNG wire#powerrail
      { S7_Templates := "SrcType := Int" } LE_Contact(in1 := "DataDI"."Konik 2 Üretim Sayac Hızı", in2 := 0)
      wire#w2
      Move(in := 0, out1 => "DataDI"."Konik 2 Üretim Sayac Hızı")
   END_RUNG
   RUNG wire#powerrail
      { S7_Templates := "SrcType := Int" } GT_Contact(in1 := "DataDI"."Konik 2 Üretim Sayac Hızı", in2 := 200)
   END_RUNG wire#w2
   RUNG wire#powerrail
      { S7_Templates := "SrcType := Int" } LE_Contact(in1 := "DataDI"."Konik 3 Üretim Sayac Hızı", in2 := 0)
      wire#w3
      Move(in := 0, out1 => "DataDI"."Konik 3 Üretim Sayac Hızı")
   END_RUNG
   RUNG wire#powerrail
      { S7_Templates := "SrcType := Int" } GT_Contact(in1 := "DataDI"."Konik 3 Üretim Sayac Hızı", in2 := 200)
   END_RUNG wire#w3
   RUNG wire#powerrail
      { S7_Templates := "SrcType := Int" } LE_Contact(in1 := "DataDI"."Konik 4 Üretim Sayac Hızı", in2 := 0)
      wire#w4
      Move(in := 0, out1 => "DataDI"."Konik 4 Üretim Sayac Hızı")
   END_RUNG
   RUNG wire#powerrail
      { S7_Templates := "SrcType := Int" } GT_Contact(in1 := "DataDI"."Konik 4 Üretim Sayac Hızı", in2 := 200)
   END_RUNG wire#w4
   RUNG wire#powerrail
      { S7_Templates := "SrcType := Int" } LE_Contact(in1 := "DataDI"."Konik 5 Üretim Sayac Hızı", in2 := 0)
      wire#w5
      Move(in := 0, out1 => "DataDI"."Konik 5 Üretim Sayac Hızı")
   END_RUNG
   RUNG wire#powerrail
      { S7_Templates := "SrcType := Int" } GT_Contact(in1 := "DataDI"."Konik 5 Üretim Sayac Hızı", in2 := 200)
   END_RUNG wire#w5
   // the same network as SCL:
   IF ("DataDI"."Konik 1 Üretim Sayac Hızı" <= 0) OR ("DataDI"."Konik 1 Üretim Sayac Hızı" > 200) THEN
       "DataDI"."Konik 1 Üretim Sayac Hızı" := 0;
   END_IF;
   IF ("DataDI"."Konik 2 Üretim Sayac Hızı" <= 0) OR ("DataDI"."Konik 2 Üretim Sayac Hızı" > 200) THEN
       "DataDI"."Konik 2 Üretim Sayac Hızı" := 0;
   END_IF;
   IF ("DataDI"."Konik 3 Üretim Sayac Hızı" <= 0) OR ("DataDI"."Konik 3 Üretim Sayac Hızı" > 200) THEN
       "DataDI"."Konik 3 Üretim Sayac Hızı" := 0;
   END_IF;
   IF ("DataDI"."Konik 4 Üretim Sayac Hızı" <= 0) OR ("DataDI"."Konik 4 Üretim Sayac Hızı" > 200) THEN
       "DataDI"."Konik 4 Üretim Sayac Hızı" := 0;
   END_IF;
   IF ("DataDI"."Konik 5 Üretim Sayac Hızı" <= 0) OR ("DataDI"."Konik 5 Üretim Sayac Hızı" > 200) THEN
       "DataDI"."Konik 5 Üretim Sayac Hızı" := 0;
   END_IF;
END_REGION
END_FUNCTION

FUNCTION "SayacRST" : Void   // FC4, LAD
{ S7_Optimized_Access := 'TRUE' }
VERSION : 0.1
   VAR_TEMP   // added for the SCL form of the ladder/FBD networks
      _w1 : Bool;
      _w2 : Bool;
      _w3 : Bool;
      _w4 : Bool;
      _w5 : Bool;
   END_VAR
BEGIN

REGION Network 1: Sayac RST
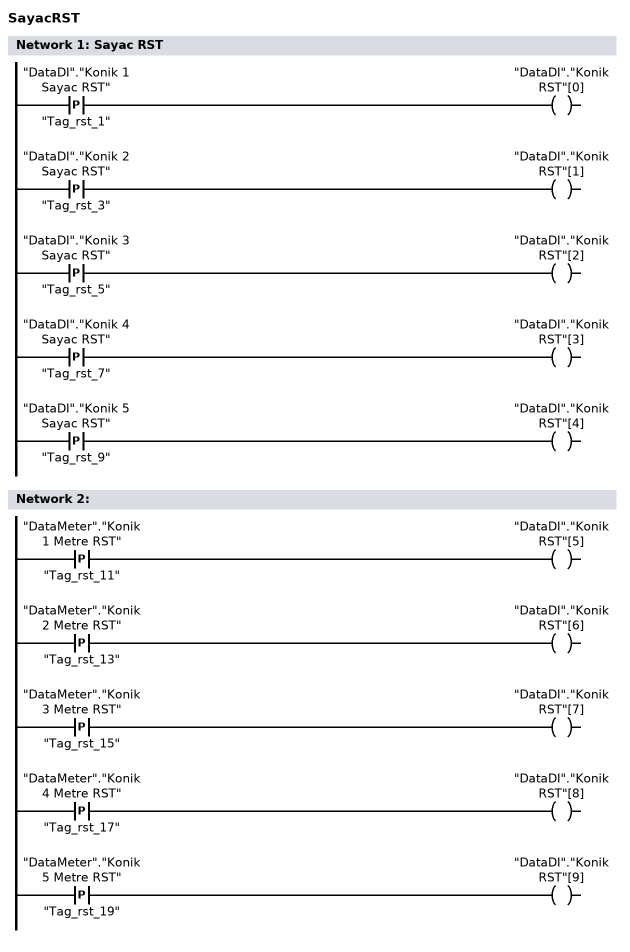
   RUNG wire#powerrail
      P_Contact(operand := "DataDI"."Konik 1 Sayac RST", bit := "Tag_rst_1")
      Coil( "DataDI"."Konik RST"[0] )
   END_RUNG
   RUNG wire#powerrail
      P_Contact(operand := "DataDI"."Konik 2 Sayac RST", bit := "Tag_rst_3")
      Coil( "DataDI"."Konik RST"[1] )
   END_RUNG
   RUNG wire#powerrail
      P_Contact(operand := "DataDI"."Konik 3 Sayac RST", bit := "Tag_rst_5")
      Coil( "DataDI"."Konik RST"[2] )
   END_RUNG
   RUNG wire#powerrail
      P_Contact(operand := "DataDI"."Konik 4 Sayac RST", bit := "Tag_rst_7")
      Coil( "DataDI"."Konik RST"[3] )
   END_RUNG
   RUNG wire#powerrail
      P_Contact(operand := "DataDI"."Konik 5 Sayac RST", bit := "Tag_rst_9")
      Coil( "DataDI"."Konik RST"[4] )
   END_RUNG
   // the same network as SCL:
   #_w1 := "DataDI"."Konik 1 Sayac RST" AND NOT "Tag_rst_1";   // rising edge of "DataDI"."Konik 1 Sayac RST"
   "Tag_rst_1" := "DataDI"."Konik 1 Sayac RST";
   "DataDI"."Konik RST"[0] := #_w1;
   #_w2 := "DataDI"."Konik 2 Sayac RST" AND NOT "Tag_rst_3";   // rising edge of "DataDI"."Konik 2 Sayac RST"
   "Tag_rst_3" := "DataDI"."Konik 2 Sayac RST";
   "DataDI"."Konik RST"[1] := #_w2;
   #_w3 := "DataDI"."Konik 3 Sayac RST" AND NOT "Tag_rst_5";   // rising edge of "DataDI"."Konik 3 Sayac RST"
   "Tag_rst_5" := "DataDI"."Konik 3 Sayac RST";
   "DataDI"."Konik RST"[2] := #_w3;
   #_w4 := "DataDI"."Konik 4 Sayac RST" AND NOT "Tag_rst_7";   // rising edge of "DataDI"."Konik 4 Sayac RST"
   "Tag_rst_7" := "DataDI"."Konik 4 Sayac RST";
   "DataDI"."Konik RST"[3] := #_w4;
   #_w5 := "DataDI"."Konik 5 Sayac RST" AND NOT "Tag_rst_9";   // rising edge of "DataDI"."Konik 5 Sayac RST"
   "Tag_rst_9" := "DataDI"."Konik 5 Sayac RST";
   "DataDI"."Konik RST"[4] := #_w5;
END_REGION

REGION Network 2
   RUNG wire#powerrail
      P_Contact(operand := "DataMeter"."Konik 1 Metre RST", bit := "Tag_rst_11")
      Coil( "DataDI"."Konik RST"[5] )
   END_RUNG
   RUNG wire#powerrail
      P_Contact(operand := "DataMeter"."Konik 2 Metre RST", bit := "Tag_rst_13")
      Coil( "DataDI"."Konik RST"[6] )
   END_RUNG
   RUNG wire#powerrail
      P_Contact(operand := "DataMeter"."Konik 3 Metre RST", bit := "Tag_rst_15")
      Coil( "DataDI"."Konik RST"[7] )
   END_RUNG
   RUNG wire#powerrail
      P_Contact(operand := "DataMeter"."Konik 4 Metre RST", bit := "Tag_rst_17")
      Coil( "DataDI"."Konik RST"[8] )
   END_RUNG
   RUNG wire#powerrail
      P_Contact(operand := "DataMeter"."Konik 5 Metre RST", bit := "Tag_rst_19")
      Coil( "DataDI"."Konik RST"[9] )
   END_RUNG
   // the same network as SCL:
   #_w1 := "DataMeter"."Konik 1 Metre RST" AND NOT "Tag_rst_11";   // rising edge of "DataMeter"."Konik 1 Metre RST"
   "Tag_rst_11" := "DataMeter"."Konik 1 Metre RST";
   "DataDI"."Konik RST"[5] := #_w1;
   #_w2 := "DataMeter"."Konik 2 Metre RST" AND NOT "Tag_rst_13";   // rising edge of "DataMeter"."Konik 2 Metre RST"
   "Tag_rst_13" := "DataMeter"."Konik 2 Metre RST";
   "DataDI"."Konik RST"[6] := #_w2;
   #_w3 := "DataMeter"."Konik 3 Metre RST" AND NOT "Tag_rst_15";   // rising edge of "DataMeter"."Konik 3 Metre RST"
   "Tag_rst_15" := "DataMeter"."Konik 3 Metre RST";
   "DataDI"."Konik RST"[7] := #_w3;
   #_w4 := "DataMeter"."Konik 4 Metre RST" AND NOT "Tag_rst_17";   // rising edge of "DataMeter"."Konik 4 Metre RST"
   "Tag_rst_17" := "DataMeter"."Konik 4 Metre RST";
   "DataDI"."Konik RST"[8] := #_w4;
   #_w5 := "DataMeter"."Konik 5 Metre RST" AND NOT "Tag_rst_19";   // rising edge of "DataMeter"."Konik 5 Metre RST"
   "Tag_rst_19" := "DataMeter"."Konik 5 Metre RST";
   "DataDI"."Konik RST"[9] := #_w5;
END_REGION
END_FUNCTION

FUNCTION "CalcMeter" : Void   // FC5, LAD
{ S7_Optimized_Access := 'TRUE' }
VERSION : 0.1
   VAR_INPUT
      EncCounter : UDInt;
      diameter : Real;
      EncResulation : Int;
   END_VAR
   VAR_OUTPUT
      Meter : UDInt;
      Realmetervalue : Real;
   END_VAR
   VAR_TEMP
      EncValue : Real;
      RealMeter : Real;
   END_VAR
BEGIN

REGION Network 1
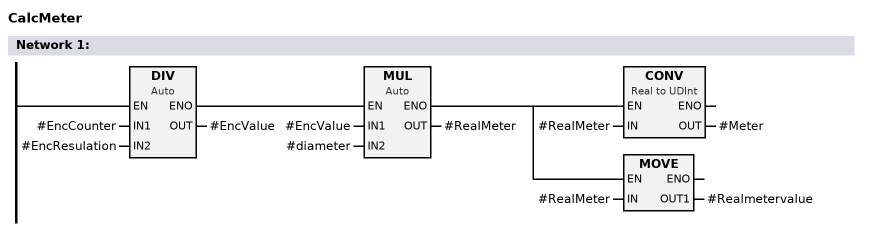
   RUNG wire#powerrail
      Div(in1 := #EncCounter, in2 := #EncResulation, out => #EncValue)
      Mul(in1 := #EncValue, in2 := #diameter, out => #RealMeter)
      wire#w1
      { S7_Templates := "[SrcType := Real, DestType := UDInt]" } Convert(in := #RealMeter, out => #Meter)
   END_RUNG
   RUNG wire#w1
      Move(in := #RealMeter, out1 => #Realmetervalue)
   END_RUNG
   // the same network as SCL:
   #EncValue := #EncCounter / #EncResulation;
   #RealMeter := #EncValue * #diameter;
   #Meter := REAL_TO_UDINT(#RealMeter);
   #Realmetervalue := #RealMeter;
END_REGION
END_FUNCTION

FUNCTION "DataTransform" : Void   // FC6, SCL
{ S7_Optimized_Access := 'TRUE' }
VERSION : 0.1
BEGIN
   "DataSendDI"."Konik 1 Üretim sayacı" := UDINT_TO_REAL("DataDI"."Konik 1 Üretim sayacı");
   "DataSendDI"."Konik 2 Üretim sayacı" := UDINT_TO_REAL("DataDI"."Konik 2 Üretim sayacı");
   "DataSendDI"."Konik 3 Üretim sayacı" := UDINT_TO_REAL("DataDI"."Konik 3 Üretim sayacı");
   "DataSendDI"."Konik 4 Üretim sayacı" := UDINT_TO_REAL("DataDI"."Konik 4 Üretim sayacı");
   "DataSendDI"."Konik 5 Üretim sayacı" := UDINT_TO_REAL("DataDI"."Konik 5 Üretim sayacı");

   "DataSendDI"."Konik 1 Besleme Run Sinyal" := "DataDI"."Konik 1 Besleme Run Sinyal";
   "DataSendDI"."Konik 2 Besleme Run Sinyal" := "DataDI"."Konik 2 Besleme Run Sinyal";
   "DataSendDI"."Konik 3  BeslemeRun Sinyal" := "DataDI"."Konik 3  BeslemeRun Sinyal";
   "DataSendDI"."Konik 4  BeslemeRun Sinyal" := "DataDI"."Konik 4  BeslemeRun Sinyal";
   "DataSendDI"."Konik 5  BeslemeRun Sinyal" := "DataDI"."Konik 5  BeslemeRun Sinyal";

   "DataSendDI"."Konik 1 Run Sinyal" := "DataDI"."Konik 1 Run Sinyal";
   "DataSendDI"."Konik 2 Run Sinyal" := "DataDI"."Konik 2 Run Sinyal";
   "DataSendDI"."Konik 3 Run Sinyal" := "DataDI"."Konik 3 Run Sinyal";
   "DataSendDI"."Konik 4 Run Sinyal" := "DataDI"."Konik 4 Run Sinyal";
   "DataSendDI"."Konik 5 Run Sinyal" := "DataDI"."Konik 5 Run Sinyal";

   "DataSendDI"."Konik 1 Üretim Sayac Hızı" := INT_TO_REAL("DataDI"."Konik 1 Üretim Sayac Hızı");
   "DataSendDI"."Konik 2 Üretim Sayac Hızı" := INT_TO_REAL("DataDI"."Konik 2 Üretim Sayac Hızı");
   "DataSendDI"."Konik 3 Üretim Sayac Hızı" := INT_TO_REAL("DataDI"."Konik 3 Üretim Sayac Hızı");
   "DataSendDI"."Konik 4 Üretim Sayac Hızı" := INT_TO_REAL("DataDI"."Konik 4 Üretim Sayac Hızı");
   "DataSendDI"."Konik 5 Üretim Sayac Hızı" := INT_TO_REAL("DataDI"."Konik 5 Üretim Sayac Hızı");

   "DataSendDI"."Konik 1 Metre Sayac" := UDINT_TO_REAL("DataMeter"."Konik 1 Metre Sayac");
   "DataSendDI"."Konik 2 Metre Sayac" := UDINT_TO_REAL("DataMeter"."Konik 2 Metre Sayac");
   "DataSendDI"."Konik 3 Metre Sayac" := UDINT_TO_REAL("DataMeter"."Konik 3 Metre Sayac");
   "DataSendDI"."Konik 4 Metre Sayac" := UDINT_TO_REAL("DataMeter"."Konik 4 Metre Sayac");
   "DataSendDI"."Konik 5 Metre Sayac" := UDINT_TO_REAL("DataMeter"."Konik 5 Metre Sayac");

   "DataSendDI"."Konik 1 Hız" := "DataMeter"."Konik 1 Hız";
   "DataSendDI"."Konik 2 Hız" := "DataMeter"."Konik 2 Hız";
   "DataSendDI"."Konik 3 Hız" := "DataMeter"."Konik 3 Hız";
   "DataSendDI"."Konik 4 Hız" := "DataMeter"."Konik 4 Hız";
   "DataSendDI"."Konik 5 Hız" := "DataMeter"."Konik 5 Hız";

   "DataMeter"."Konik 1 Metre RST" := "DataSendDI"."Konik 1 Metre RST";
   "DataMeter"."Konik 2 Metre RST" := "DataSendDI"."Konik 2 Metre RST";
   "DataMeter"."Konik 3 Metre RST" := "DataSendDI"."Konik 3 Metre RST";
   "DataMeter"."Konik 4 Metre RST" := "DataSendDI"."Konik 4 Metre RST";
   "DataMeter"."Konik 5 Metre RST" := "DataSendDI"."Konik 5 Metre RST";

   "DataDI"."Konik 1 Sayac RST" := "DataSendDI"."Konik 1 Sayac RST";
   "DataDI"."Konik 2 Sayac RST" := "DataSendDI"."Konik 2 Sayac RST";
   "DataDI"."Konik 3 Sayac RST" := "DataSendDI"."Konik 3 Sayac RST";
   "DataDI"."Konik 4 Sayac RST" := "DataSendDI"."Konik 4 Sayac RST";
   "DataDI"."Konik 5 Sayac RST" := "DataSendDI"."Konik 5 Sayac RST";
END_FUNCTION

ORGANIZATION_BLOCK "Main"   // OB1, LAD, ProgramCycle
TITLE = "Main Program Sweep (Cycle)"
{ S7_Optimized_Access := 'TRUE' }
VERSION : 0.1
   VAR_INPUT
      Initial_Call : Bool;   // Initial call of this OB
      Remanence : Bool;   // =True, if remanent data are available
   END_VAR
   VAR_TEMP
      timerout : Bool;
   END_VAR
BEGIN

REGION Network 1
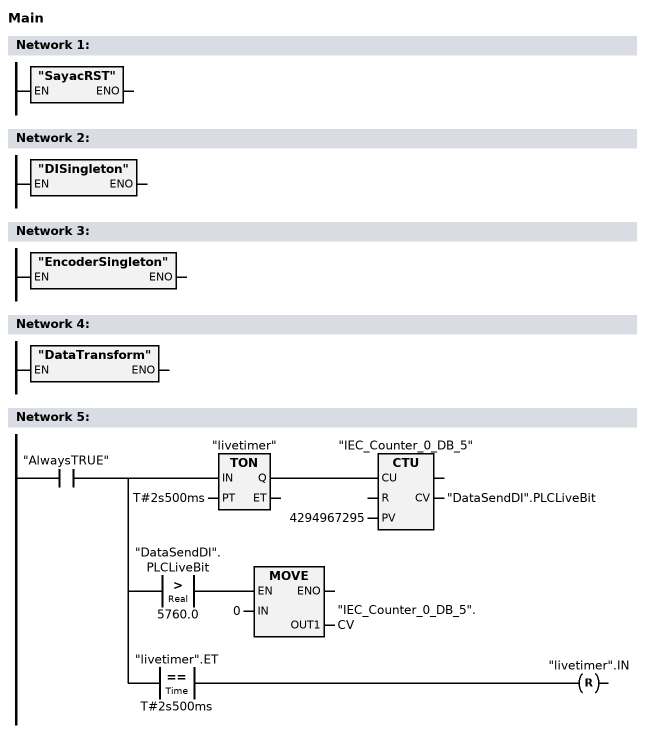
   RUNG wire#powerrail
      "SayacRST"()
   END_RUNG
   // the same network as SCL:
   "SayacRST"();
END_REGION

REGION Network 2
   RUNG wire#powerrail
      "DISingleton"()
   END_RUNG
   // the same network as SCL:
   "DISingleton"();
END_REGION

REGION Network 3
   RUNG wire#powerrail
      "EncoderSingleton"()
   END_RUNG
   // the same network as SCL:
   "EncoderSingleton"();
END_REGION

REGION Network 4
   RUNG wire#powerrail
      "DataTransform"()
   END_RUNG
   // the same network as SCL:
   "DataTransform"();
END_REGION

REGION Network 5
   "livetimer".TON(IN := "AlwaysTRUE", PT := T#2s500ms);
   "IEC_Counter_0_DB_5".CTU(CU := "livetimer".Q, PV := 4294967295, CV => "DataSendDI".PLCLiveBit);
   IF "AlwaysTRUE" AND ("DataSendDI".PLCLiveBit > 5760.0) THEN "IEC_Counter_0_DB_5".CV := 0; END_IF;
   IF "AlwaysTRUE" AND ("livetimer".ET = T#2s500ms) THEN "livetimer".IN := FALSE; END_IF;
END_REGION
END_ORGANIZATION_BLOCK